//{attribute 'qualified_only'}
VAR_GLOBAL
	bRelaisBoiler 		AT %Q*	: BOOL;	(* Geschakeld stopcontact *)
END_VAR

(* stored: Version 1.1.0.1
   GVL GVL_Boiler: Id {9f6c2382-8539-464b-a74f-a60f632b839b} *)
